FUNCTION_BLOCK IA_RHS (* ISOBUS Adapter for Rear Hitch Status (RHS) *)
  (* Standard: ISO 11783-7; Classification: PGN 65093; Description: Copyright (c) 2024-2026 HR Agrartechnik GmbH This program and the accompanying materials are made available under the terms of the Eclipse Public License 2.0 which is available at https://www.eclipse.org/legal/epl-2.0/ SPDX-License-Identifier: EPL-2.0 *)
  (* Version 1.0, 2026-04-19, Franz Höpfinger, HR Agrartechnik GmbH, initial API and implementation (Adapter Wrapper for I_RHS) *)
  PACKAGE isobus::tecu;
  IMPORT eclipse4diac::core::TypeHash;
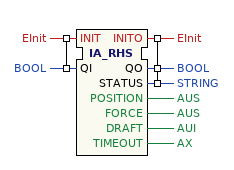
  EVENT_INPUT
    INIT : EInit WITH QI; (* Service Initialization *)
  END_EVENT
  EVENT_OUTPUT
    INITO : EInit WITH QO, STATUS; (* Initialization Confirm *)
  END_EVENT
  VAR_INPUT
    QI : BOOL; (* Event Input Qualifier *)
  END_VAR
  VAR_OUTPUT
    QO : BOOL; (* Event Output Qualifier *)
    STATUS : STRING;
  END_VAR
  PLUGS
    POSITION : adapter::types::unidirectional::AUS; (* Rear Hitch Position *)
    FORCE : adapter::types::unidirectional::AUS; (* Rear Nominal Lower Link Force *)
    DRAFT : adapter::types::unidirectional::AUI; (* Rear Draft *)
    TIMEOUT : adapter::types::unidirectional::AX; (* Timeout Status *)
  END_PLUGS
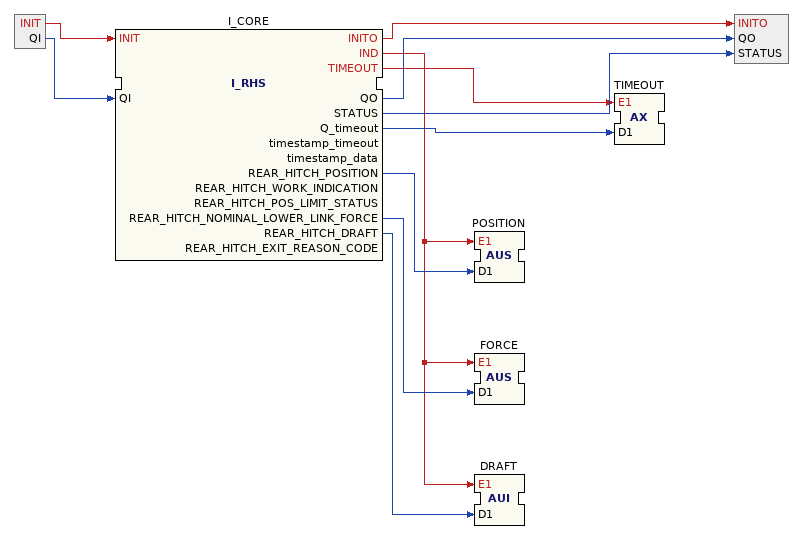
  FBS
    I_CORE : isobus::tecu::I_RHS;
  END_FBS
  EVENT_CONNECTIONS
    INIT TO I_CORE.INIT;
    I_CORE.INITO TO INITO;
    I_CORE.IND TO POSITION.E1;
    I_CORE.IND TO FORCE.E1;
    I_CORE.IND TO DRAFT.E1;
    I_CORE.TIMEOUT TO TIMEOUT.E1;
  END_CONNECTIONS
  DATA_CONNECTIONS
    QI TO I_CORE.QI;
    I_CORE.QO TO QO;
    I_CORE.STATUS TO STATUS;
    I_CORE.REAR_HITCH_POSITION TO POSITION.D1;
    I_CORE.REAR_HITCH_NOMINAL_LOWER_LINK_FORCE TO FORCE.D1;
    I_CORE.REAR_HITCH_DRAFT TO DRAFT.D1;
    I_CORE.Q_timeout TO TIMEOUT.D1;
  END_CONNECTIONS
END_FUNCTION_BLOCK
